FUNCTION_BLOCK FB_DirectoryContorlTest EXTENDS TcUnit.FB_TestSuite

CreateDictionaryTest();

METHOD CreateDictionaryTest
VAR_INPUT
END_VAR

VAR_INST
	Timer : TON := (PT := T#50S);
	fbDirectoryControl : FB_DirectoryControl;
	bDone : REFERENCE TO BOOL;
END_VAR
IF TEST_ORDERED('CreateDiectionaryTest') THEN
	Timer(In:=TRUE);
	
	
	IF Timer.Q THEN
		
		AssertEquals(Expected := bDone
					,Actual := bDone
					,Message := 'CreateDirectoryFail' );
	
		TEST_FINISHED();
	END_IF
END_IF
END_METHOD

END_FUNCTION_BLOCK

(* stored: Version 1.1.0.1, ProductVersion 3.1.4024.12
   POU FB_DirectoryContorlTest: Id {82fe1301-1a45-494b-9089-8d51e5aaed18}, SpecialFunc None
   Method CreateDictionaryTest: Id {2a402643-5da0-470f-ab5b-f1f8ca379479} *)
